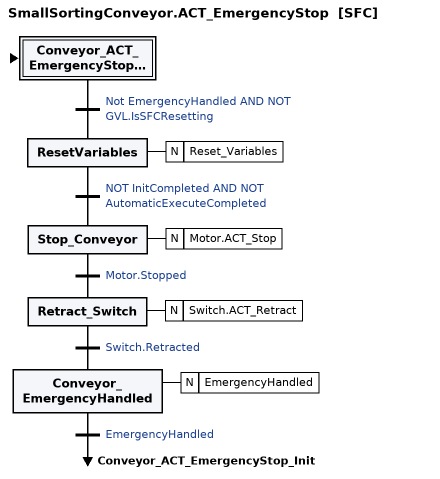
INITIAL_STEP Conveyor_ACT_EmergencyStop_Init:
END_STEP
TRANSITION FROM Conveyor_ACT_EmergencyStop_Init TO ResetVariables
  := Not EmergencyHandled AND NOT GVL.IsSFCResetting;
END_TRANSITION
STEP ResetVariables:
  Reset_Variables(N);
END_STEP
TRANSITION FROM ResetVariables TO Stop_Conveyor
  := NOT InitCompleted AND NOT AutomaticExecuteCompleted;
END_TRANSITION
STEP Stop_Conveyor:
  Motor.ACT_Stop(N);
END_STEP
TRANSITION FROM Stop_Conveyor TO Retract_Switch
  := Motor.Stopped;
END_TRANSITION
STEP Retract_Switch:
  Switch.ACT_Retract(N);
END_STEP
TRANSITION FROM Retract_Switch TO Conveyor_EmergencyHandled
  := Switch.Retracted;
END_TRANSITION
STEP Conveyor_EmergencyHandled:
  EmergencyHandled(N);
END_STEP
TRANSITION FROM Conveyor_EmergencyHandled TO Conveyor_ACT_EmergencyStop_Init
  := EmergencyHandled;
END_TRANSITION
END_ACTION

ACTION ACT_Init:
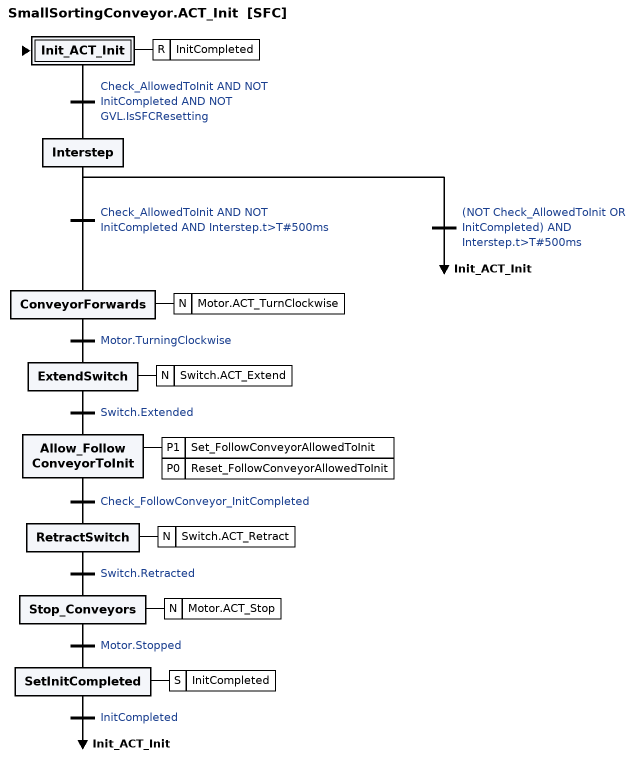
INITIAL_STEP Init_ACT_Init:
  InitCompleted(R);
END_STEP
TRANSITION FROM Init_ACT_Init TO Interstep
  := Check_AllowedToInit AND NOT InitCompleted AND NOT GVL.IsSFCResetting;
END_TRANSITION
STEP Interstep:
END_STEP
TRANSITION FROM Interstep TO ConveyorForwards
  := Check_AllowedToInit AND NOT InitCompleted AND Interstep.t>T#500ms;
END_TRANSITION
TRANSITION FROM Interstep TO Init_ACT_Init
  := (NOT Check_AllowedToInit OR InitCompleted) AND Interstep.t>T#500ms;
END_TRANSITION
STEP ConveyorForwards:
  Motor.ACT_TurnClockwise(N);
END_STEP
TRANSITION FROM ConveyorForwards TO ExtendSwitch
  := Motor.TurningClockwise;
END_TRANSITION
STEP ExtendSwitch:
  Switch.ACT_Extend(N);
END_STEP
TRANSITION FROM ExtendSwitch TO Allow_FollowConveyorToInit
  := Switch.Extended;
END_TRANSITION
STEP Allow_FollowConveyorToInit:
  Set_FollowConveyorAllowedToInit(P1);
  Reset_FollowConveyorAllowedToInit(P0);
END_STEP
TRANSITION FROM Allow_FollowConveyorToInit TO RetractSwitch
  := Check_FollowConveyor_InitCompleted;
END_TRANSITION
STEP RetractSwitch:
  Switch.ACT_Retract(N);
END_STEP
TRANSITION FROM RetractSwitch TO Stop_Conveyors
  := Switch.Retracted;
END_TRANSITION
STEP Stop_Conveyors:
  Motor.ACT_Stop(N);
END_STEP
TRANSITION FROM Stop_Conveyors TO SetInitCompleted
  := Motor.Stopped;
END_TRANSITION
STEP SetInitCompleted:
  InitCompleted(S);
END_STEP
TRANSITION FROM SetInitCompleted TO Init_ACT_Init
  := InitCompleted;
END_TRANSITION
END_ACTION
END_FUNCTION_BLOCK

FUNCTION_BLOCK Stack
VAR_INPUT	
	//Hardware
	Seperator : MonostableCylinder;
	Panel : OperationPanel;	
	WPAvailable : MicroSwitch;
	InductiveSensor : InductiveSensor;
	OpticalSensor : OpticalSensor;
	WeightModule : WeightModule;
	
	//Software
	Check_WPPickedUp : BOOL;
	SFCReset : BOOL;	//Only for SFC implementation
END_VAR
VAR_OUTPUT	
	//Software
	StartButton : BOOL;
	ManuelMode : BOOL;
	AutomaticMode : BOOL;
	InitCompleted : BOOL;
	AutomaticExecuteCompleted : BOOL;
	EmergencyStop : BOOL;
	EmergencyHandled : BOOL;	
	
END_VAR
VAR	
	//Software
	WPProvided : BOOL;	
	WPType_White : BOOL;
	WPType_Black : BOOL;
	WPType_Metallic : BOOL;	
	WPWeight_Light : BOOL;
	WPWeight_Medium : BOOL;
	WPWeight_Heavy : BOOL;	
	Timer : TON;	
END_VAR

                  Panel();
StartButton := Panel.StartButton;
ManuelMode := Panel.ManuelMode; 
AutomaticMode := Panel.AutomaticMode;
EmergencyStop := Panel.EmergencyStop;
Check_WPPickedUp := Main.Check_Stack_WPPickedUp;
                

ACTION Reset_Timer:
                      Timer(IN:=FALSE);
                    
END_ACTION

ACTION Reset_Variables:
                      InitCompleted := FALSE;
AutomaticExecuteCompleted := FALSE;

WPType_White:=FALSE;
WPType_Black:=FALSE;
WPType_Metallic:=FALSE;
WPWeight_Light:=FALSE;
WPWeight_Medium:=FALSE;
WPWeight_Heavy:=FALSE;
                    
END_ACTION

ACTION Set_Timer250ms:
                      Timer(IN:=TRUE, PT:=T#250MS);
                    
END_ACTION

ACTION Set_WPParameters_AND_WPProvided:
                      //WPType
IF(NOT InductiveSensor.DI_WPMetallic AND NOT OpticalSensor.DI_WPLight)THEN
	WPType_Black:=TRUE;
	WPType_White:=FALSE;
	WPType_Metallic:=FALSE;
ELSIF(NOT InductiveSensor.DI_WPMetallic AND OpticalSensor.DI_WPLight)THEN
	WPType_Black:=FALSE;
	WPType_White:=TRUE;
	WPType_Metallic:=FALSE;
ELSIF(InductiveSensor.DI_WPMetallic)THEN
	WPType_Black:=FALSE;
	WPType_White:=FALSE;
	WPType_Metallic:=TRUE;
END_IF
//WPWeight
IF(WeightModule.AI_WPWeight<12000)THEN
	WPWeight_Light:=TRUE;
	WPWeight_Medium:=FALSE;
	WPWeight_Heavy:=FALSE;
ELSIF(12000<=WeightModule.AI_WPWeight AND WeightModule.AI_WPWeight<24000)THEN
	WPWeight_Light:=FALSE;
	WPWeight_Medium:=TRUE;
	WPWeight_Heavy:=FALSE;
ELSIF(2400<=WeightModule.AI_WPWeight)THEN
	WPWeight_Light:=FALSE;
	WPWeight_Medium:=FALSE;
	WPWeight_Heavy:=TRUE;	
END_IF

WPProvided:=TRUE;
                    
END_ACTION

ACTION ACT_ProvideWP:
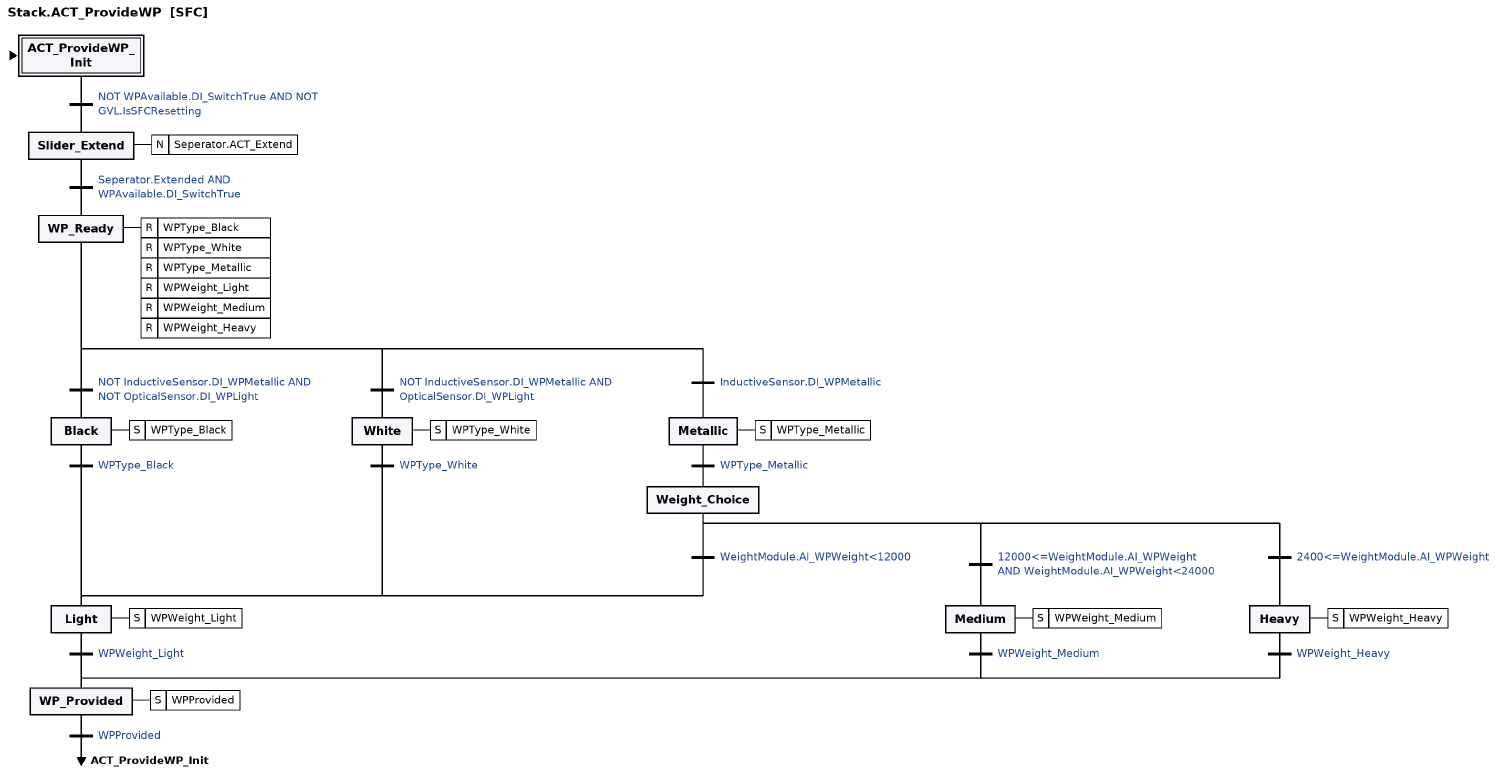
INITIAL_STEP ACT_ProvideWP_Init:
END_STEP
TRANSITION FROM ACT_ProvideWP_Init TO Slider_Extend
  := NOT WPAvailable.DI_SwitchTrue AND NOT GVL.IsSFCResetting;
END_TRANSITION
STEP Slider_Extend:
  Seperator.ACT_Extend(N);
END_STEP
TRANSITION FROM Slider_Extend TO WP_Ready
  := Seperator.Extended AND WPAvailable.DI_SwitchTrue;
END_TRANSITION
STEP WP_Ready:
  WPType_Black(R);
  WPType_White(R);
  WPType_Metallic(R);
  WPWeight_Light(R);
  WPWeight_Medium(R);
  WPWeight_Heavy(R);
END_STEP
TRANSITION FROM WP_Ready TO Black
  := NOT InductiveSensor.DI_WPMetallic AND NOT OpticalSensor.DI_WPLight;
END_TRANSITION
TRANSITION FROM WP_Ready TO White
  := NOT InductiveSensor.DI_WPMetallic AND OpticalSensor.DI_WPLight;
END_TRANSITION
TRANSITION FROM WP_Ready TO Metallic
  := InductiveSensor.DI_WPMetallic;
END_TRANSITION
STEP Black:
  WPType_Black(S);
END_STEP
TRANSITION FROM Black TO Light
  := WPType_Black;
END_TRANSITION
STEP Light:
  WPWeight_Light(S);
END_STEP
TRANSITION FROM Light TO WP_Provided
  := WPWeight_Light;
END_TRANSITION
STEP White:
  WPType_White(S);
END_STEP
TRANSITION FROM White TO Light
  := WPType_White;
END_TRANSITION
STEP Metallic:
  WPType_Metallic(S);
END_STEP
TRANSITION FROM Metallic TO Weight_Choice
  := WPType_Metallic;
END_TRANSITION
STEP Weight_Choice:
END_STEP
TRANSITION FROM Weight_Choice TO Light
  := WeightModule.AI_WPWeight<12000;
END_TRANSITION
TRANSITION FROM Weight_Choice TO Medium
  := 12000<=WeightModule.AI_WPWeight AND WeightModule.AI_WPWeight<24000;
END_TRANSITION
TRANSITION FROM Weight_Choice TO Heavy
  := 2400<=WeightModule.AI_WPWeight;
END_TRANSITION
STEP Medium:
  WPWeight_Medium(S);
END_STEP
TRANSITION FROM Medium TO WP_Provided
  := WPWeight_Medium;
END_TRANSITION
STEP Heavy:
  WPWeight_Heavy(S);
END_STEP
TRANSITION FROM Heavy TO WP_Provided
  := WPWeight_Heavy;
END_TRANSITION
STEP WP_Provided:
  WPProvided(S);
END_STEP
TRANSITION FROM WP_Provided TO ACT_ProvideWP_Init
  := WPProvided;
END_TRANSITION
END_ACTION

ACTION ACT_AutomaticExecute:
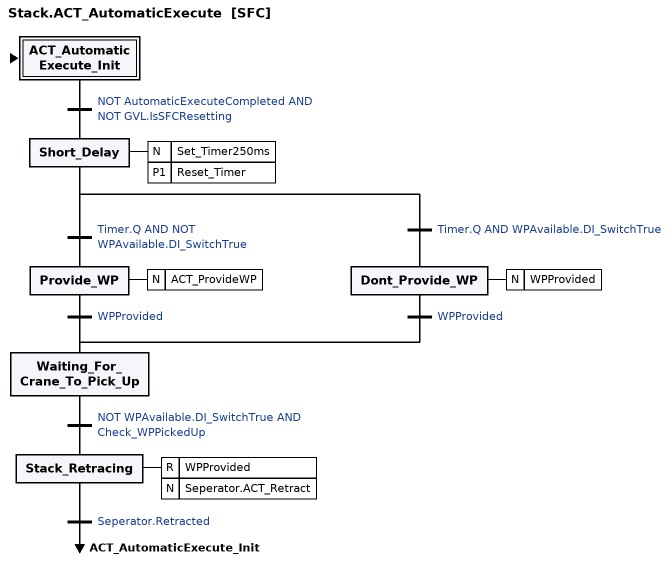
INITIAL_STEP ACT_AutomaticExecute_Init:
END_STEP
TRANSITION FROM ACT_AutomaticExecute_Init TO Short_Delay
  := NOT AutomaticExecuteCompleted AND NOT GVL.IsSFCResetting;
END_TRANSITION
STEP Short_Delay:
  Set_Timer250ms(N);
  Reset_Timer(P1);
END_STEP
TRANSITION FROM Short_Delay TO Provide_WP
  := Timer.Q AND NOT WPAvailable.DI_SwitchTrue;
END_TRANSITION
TRANSITION FROM Short_Delay TO Dont_Provide_WP
  := Timer.Q AND WPAvailable.DI_SwitchTrue;
END_TRANSITION
STEP Provide_WP:
  ACT_ProvideWP(N);
END_STEP
TRANSITION FROM Provide_WP TO Waiting_For_Crane_To_Pick_Up
  := WPProvided;
END_TRANSITION
STEP Dont_Provide_WP:
  WPProvided(N);
END_STEP
TRANSITION FROM Dont_Provide_WP TO Waiting_For_Crane_To_Pick_Up
  := WPProvided;
END_TRANSITION
STEP Waiting_For_Crane_To_Pick_Up:
END_STEP
TRANSITION FROM Waiting_For_Crane_To_Pick_Up TO Stack_Retracing
  := NOT WPAvailable.DI_SwitchTrue AND Check_WPPickedUp;
END_TRANSITION
STEP Stack_Retracing:
  WPProvided(R);
  Seperator.ACT_Retract(N);
END_STEP
TRANSITION FROM Stack_Retracing TO ACT_AutomaticExecute_Init
  := Seperator.Retracted;
END_TRANSITION
END_ACTION

ACTION ACT_EmergencyStop:
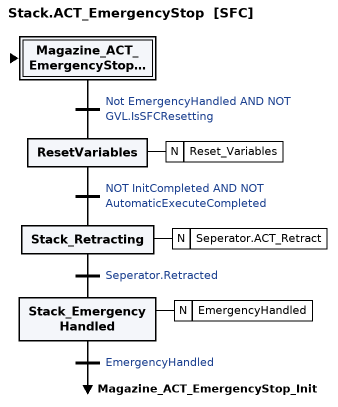
INITIAL_STEP Magazine_ACT_EmergencyStop_Init:
END_STEP
TRANSITION FROM Magazine_ACT_EmergencyStop_Init TO ResetVariables
  := Not EmergencyHandled AND NOT GVL.IsSFCResetting;
END_TRANSITION
STEP ResetVariables:
  Reset_Variables(N);
END_STEP
TRANSITION FROM ResetVariables TO Stack_Retracting
  := NOT InitCompleted AND NOT AutomaticExecuteCompleted;
END_TRANSITION
STEP Stack_Retracting:
  Seperator.ACT_Retract(N);
END_STEP
TRANSITION FROM Stack_Retracting TO Stack_EmergencyHandled
  := Seperator.Retracted;
END_TRANSITION
STEP Stack_EmergencyHandled:
  EmergencyHandled(N);
END_STEP
TRANSITION FROM Stack_EmergencyHandled TO Magazine_ACT_EmergencyStop_Init
  := EmergencyHandled;
END_TRANSITION
END_ACTION

ACTION ACT_Init:
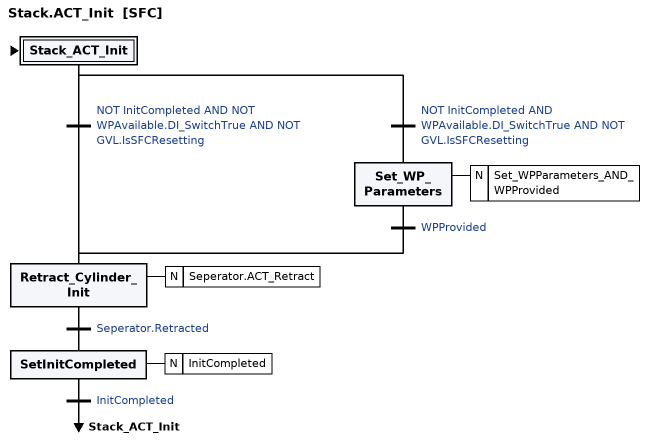
INITIAL_STEP Stack_ACT_Init:
END_STEP
TRANSITION FROM Stack_ACT_Init TO Retract_Cylinder_Init
  := NOT InitCompleted AND NOT WPAvailable.DI_SwitchTrue AND NOT GVL.IsSFCResetting;
END_TRANSITION
TRANSITION FROM Stack_ACT_Init TO Set_WP_Parameters
  := NOT InitCompleted AND WPAvailable.DI_SwitchTrue AND NOT GVL.IsSFCResetting;
END_TRANSITION
STEP Set_WP_Parameters:
  Set_WPParameters_AND_WPProvided(N);
END_STEP
TRANSITION FROM Set_WP_Parameters TO Retract_Cylinder_Init
  := WPProvided;
END_TRANSITION
STEP Retract_Cylinder_Init:
  Seperator.ACT_Retract(N);
END_STEP
TRANSITION FROM Retract_Cylinder_Init TO SetInitCompleted
  := Seperator.Retracted;
END_TRANSITION
STEP SetInitCompleted:
  InitCompleted(N);
END_STEP
TRANSITION FROM SetInitCompleted TO Stack_ACT_Init
  := InitCompleted;
END_TRANSITION
END_ACTION
END_FUNCTION_BLOCK

FUNCTION_BLOCK Stamp
VAR_INPUT
	//Hardware
	Panel : OperationPanel;
	PressureSensor : PressureSensor;
	PropValve : ProportionalValve;
	WPAvailable : MicroSwitch;
	StampingCylinder : MonostableCylinder;
	SlidingCylinder : BistableCylinder;			
	
	//Software	
	SoftwareEmergency : BOOL;
	Check_Allowed_To_Operate : BOOL;
	Check_WPWeight_Light : BOOL;
	Check_WPWeight_Medium : BOOL;
    Check_WPWeight_Heavy : BOOL;
	SFCReset : BOOL;	//Only for SFC implementation
END_VAR
VAR_OUTPUT
	//Software
	StartButton : BOOL;	
	ManuelMode : BOOL;
	AutomaticMode : BOOL;
	InitCompleted : BOOL;
	AutomaticExecuteCompleted : BOOL;
	EmergencyStop : BOOL;		
	EmergencyHandled : BOOL;
	IsStamping : BOOL;
	
END_VAR
VAR
	//Software
	WPStamped : BOOL;
	WPType_White : BOOL;
	WPType_Black : BOOL;
	WPType_Metallic : BOOL;
	WPWeight_Light : BOOL;
	WPWeight_Medium : BOOL;
	WPWeight_Heavy : BOOL;
	Timer : TON;	
END_VAR

                  Panel();
StartButton := Panel.StartButton;
ManuelMode := Panel.ManuelMode; 
AutomaticMode := Panel.AutomaticMode;
EmergencyStop := Panel.EmergencyStop;
Check_Allowed_To_Operate := Main.Check_Stamp_AllowedToOperate;
Check_WPWeight_Light:=Main.Crane_WPWeight_Light;
Check_WPWeight_Medium:=Main.Crane_WPWeight_Medium;
Check_WPWeight_Heavy:=Main.Crane_WPWeight_Heavy;
                

ACTION ExtendStampingCylinder_AND_Timer1500ms:
                      StampingCylinder.ACT_Extend();
Timer(IN:=TRUE, PT:=T#1500MS);
                    
END_ACTION

ACTION Reset_Pressure:
                      PropValve.AO_SetPressure:=0;
                    
END_ACTION

ACTION Reset_Timer:
                      Timer(IN:=FALSE);
                    
END_ACTION

ACTION Reset_Variables:
                      InitCompleted := FALSE;
AutomaticExecuteCompleted := FALSE;

propValve.AO_SetPressure:=0;
IsStamping:=FALSE;
WPStamped:=FALSE;
WPType_Black := FALSE;
WPType_White := FALSE;
WPType_Metallic := FALSE;
WPWeight_Light := FALSE;
WPWeight_Medium := FALSE;
WPWeight_Heavy := FALSE;
                    
END_ACTION

ACTION Set_HeavyPressure:
                      PropValve.AO_SetPressure:=7000;
                    
END_ACTION

ACTION Set_LightPressure:
                      PropValve.AO_SetPressure:=4000;
                    
END_ACTION

ACTION Set_MediumPressure:
                      PropValve.AO_SetPressure:=5500;
                    
END_ACTION

ACTION Set_Timer1000ms:
                      Timer(IN:=TRUE, PT:=T#1000MS);
                    
END_ACTION

ACTION Set_Timer500ms:
                      Timer(IN:=TRUE, PT:=T#500ms);
                    
END_ACTION

ACTION Set_WPWeight:
                      WPWeight_Light := Check_WPWeight_Light;
WPWeight_Medium := Check_WPWeight_Medium;
WPWeight_Heavy := Check_WPWeight_Heavy;
                    
END_ACTION

ACTION ACT_Stamp:
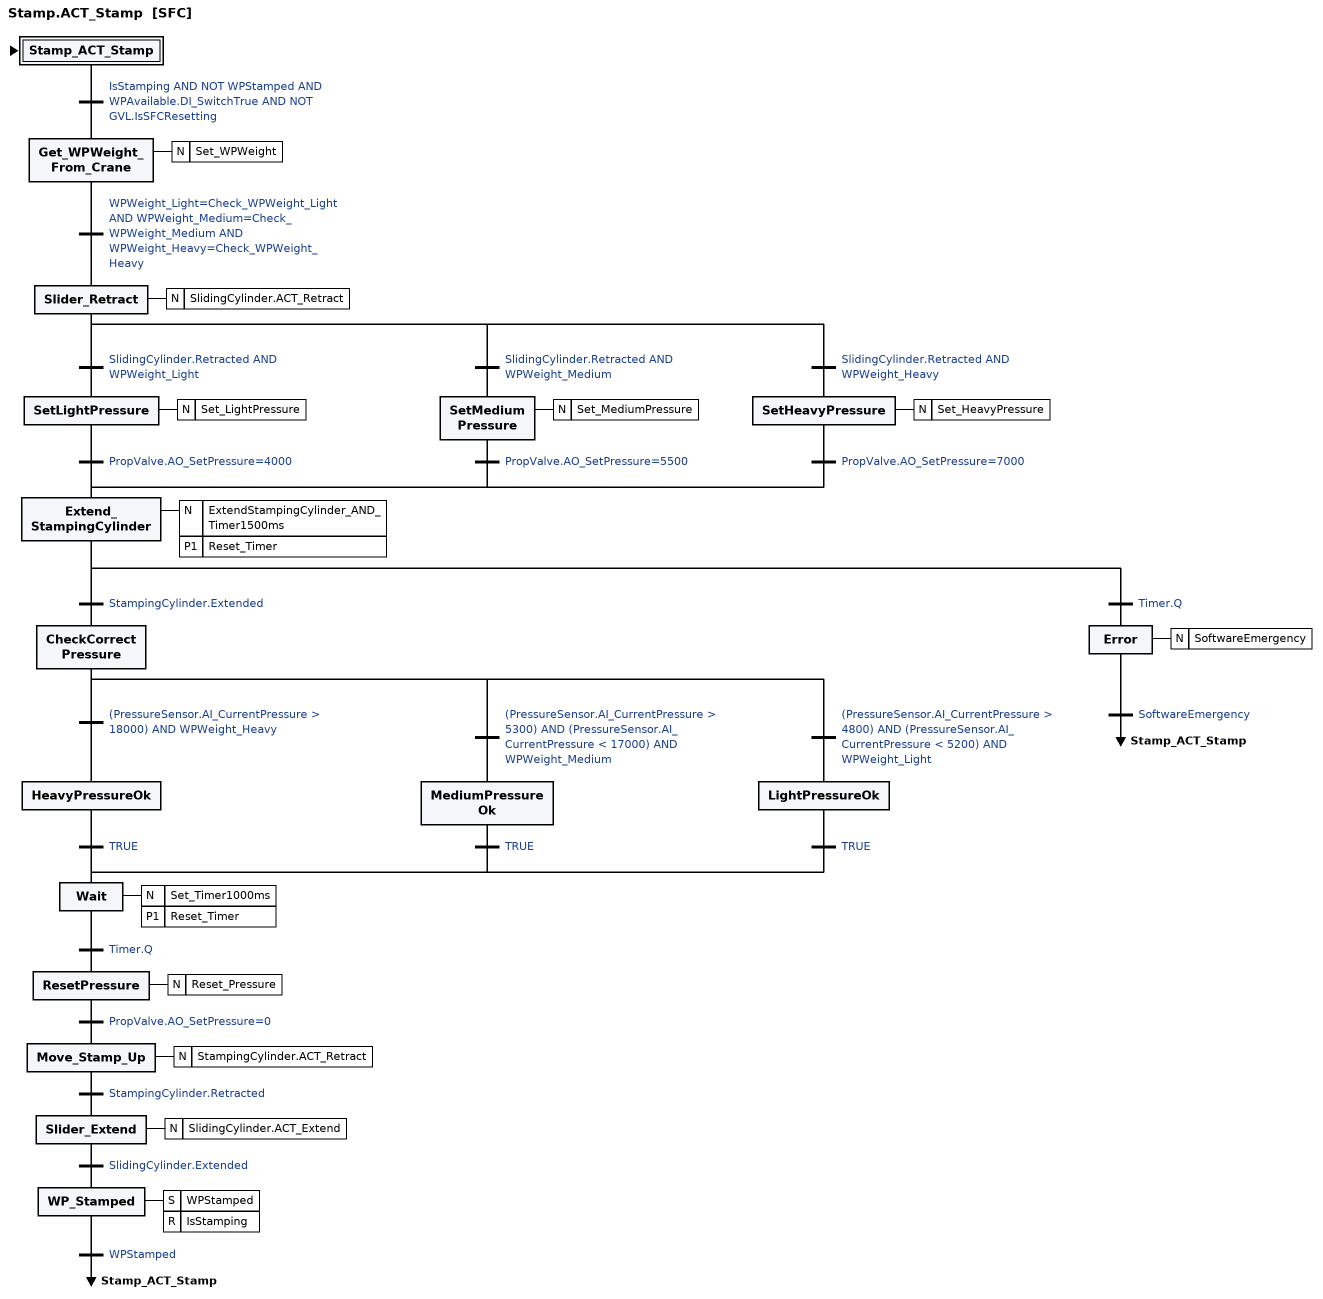
INITIAL_STEP Stamp_ACT_Stamp:
END_STEP
TRANSITION FROM Stamp_ACT_Stamp TO Get_WPWeight_From_Crane
  := IsStamping AND NOT WPStamped AND WPAvailable.DI_SwitchTrue AND NOT GVL.IsSFCResetting;
END_TRANSITION
STEP Get_WPWeight_From_Crane:
  Set_WPWeight(N);
END_STEP
TRANSITION FROM Get_WPWeight_From_Crane TO Slider_Retract
  := WPWeight_Light=Check_WPWeight_Light AND WPWeight_Medium=Check_WPWeight_Medium AND WPWeight_Heavy=Check_WPWeight_Heavy;
END_TRANSITION
STEP Slider_Retract:
  SlidingCylinder.ACT_Retract(N);
END_STEP
TRANSITION FROM Slider_Retract TO SetLightPressure
  := SlidingCylinder.Retracted AND WPWeight_Light;
END_TRANSITION
TRANSITION FROM Slider_Retract TO SetMediumPressure
  := SlidingCylinder.Retracted AND WPWeight_Medium;
END_TRANSITION
TRANSITION FROM Slider_Retract TO SetHeavyPressure
  := SlidingCylinder.Retracted AND WPWeight_Heavy;
END_TRANSITION
STEP SetLightPressure:
  Set_LightPressure(N);
END_STEP
TRANSITION FROM SetLightPressure TO Extend_StampingCylinder
  := PropValve.AO_SetPressure=4000;
END_TRANSITION
STEP SetMediumPressure:
  Set_MediumPressure(N);
END_STEP
TRANSITION FROM SetMediumPressure TO Extend_StampingCylinder
  := PropValve.AO_SetPressure=5500;
END_TRANSITION
STEP SetHeavyPressure:
  Set_HeavyPressure(N);
END_STEP
TRANSITION FROM SetHeavyPressure TO Extend_StampingCylinder
  := PropValve.AO_SetPressure=7000;
END_TRANSITION
STEP Extend_StampingCylinder:
  ExtendStampingCylinder_AND_Timer1500ms(N);
  Reset_Timer(P1);
END_STEP
TRANSITION FROM Extend_StampingCylinder TO CheckCorrectPressure
  := StampingCylinder.Extended;
END_TRANSITION
TRANSITION FROM Extend_StampingCylinder TO Error
  := Timer.Q;
END_TRANSITION
STEP CheckCorrectPressure:
END_STEP
TRANSITION FROM CheckCorrectPressure TO HeavyPressureOk
  := (PressureSensor.AI_CurrentPressure > 18000) AND WPWeight_Heavy;
END_TRANSITION
TRANSITION FROM CheckCorrectPressure TO MediumPressureOk
  := (PressureSensor.AI_CurrentPressure > 5300) AND (PressureSensor.AI_CurrentPressure < 17000) AND WPWeight_Medium;
END_TRANSITION
TRANSITION FROM CheckCorrectPressure TO LightPressureOk
  := (PressureSensor.AI_CurrentPressure > 4800) AND (PressureSensor.AI_CurrentPressure < 5200) AND WPWeight_Light;
END_TRANSITION
STEP HeavyPressureOk:
END_STEP
TRANSITION FROM HeavyPressureOk TO Wait
  := TRUE;
END_TRANSITION
STEP MediumPressureOk:
END_STEP
TRANSITION FROM MediumPressureOk TO Wait
  := TRUE;
END_TRANSITION
STEP LightPressureOk:
END_STEP
TRANSITION FROM LightPressureOk TO Wait
  := TRUE;
END_TRANSITION
STEP Error:
  SoftwareEmergency(N);
END_STEP
TRANSITION FROM Error TO Stamp_ACT_Stamp
  := SoftwareEmergency;
END_TRANSITION
STEP Wait:
  Set_Timer1000ms(N);
  Reset_Timer(P1);
END_STEP
TRANSITION FROM Wait TO ResetPressure
  := Timer.Q;
END_TRANSITION
STEP ResetPressure:
  Reset_Pressure(N);
END_STEP
TRANSITION FROM ResetPressure TO Move_Stamp_Up
  := PropValve.AO_SetPressure=0;
END_TRANSITION
STEP Move_Stamp_Up:
  StampingCylinder.ACT_Retract(N);
END_STEP
TRANSITION FROM Move_Stamp_Up TO Slider_Extend
  := StampingCylinder.Retracted;
END_TRANSITION
STEP Slider_Extend:
  SlidingCylinder.ACT_Extend(N);
END_STEP
TRANSITION FROM Slider_Extend TO WP_Stamped
  := SlidingCylinder.Extended;
END_TRANSITION
STEP WP_Stamped:
  WPStamped(S);
  IsStamping(R);
END_STEP
TRANSITION FROM WP_Stamped TO Stamp_ACT_Stamp
  := WPStamped;
END_TRANSITION
END_ACTION

ACTION ACT_AutomaticExecute:
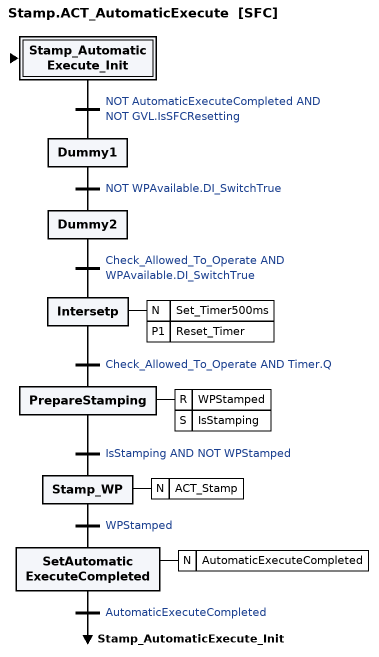
INITIAL_STEP Stamp_AutomaticExecute_Init:
END_STEP
TRANSITION FROM Stamp_AutomaticExecute_Init TO Dummy1
  := NOT AutomaticExecuteCompleted AND NOT GVL.IsSFCResetting;
END_TRANSITION
STEP Dummy1:
END_STEP
TRANSITION FROM Dummy1 TO Dummy2
  := NOT WPAvailable.DI_SwitchTrue;
END_TRANSITION
STEP Dummy2:
END_STEP
TRANSITION FROM Dummy2 TO Intersetp
  := Check_Allowed_To_Operate AND WPAvailable.DI_SwitchTrue;
END_TRANSITION
STEP Intersetp:
  Set_Timer500ms(N);
  Reset_Timer(P1);
END_STEP
TRANSITION FROM Intersetp TO PrepareStamping
  := Check_Allowed_To_Operate AND Timer.Q;
END_TRANSITION
STEP PrepareStamping:
  WPStamped(R);
  IsStamping(S);
END_STEP
TRANSITION FROM PrepareStamping TO Stamp_WP
  := IsStamping AND NOT WPStamped;
END_TRANSITION
STEP Stamp_WP:
  ACT_Stamp(N);
END_STEP
TRANSITION FROM Stamp_WP TO SetAutomaticExecuteCompleted
  := WPStamped;
END_TRANSITION
STEP SetAutomaticExecuteCompleted:
  AutomaticExecuteCompleted(N);
END_STEP
TRANSITION FROM SetAutomaticExecuteCompleted TO Stamp_AutomaticExecute_Init
  := AutomaticExecuteCompleted;
END_TRANSITION
END_ACTION

ACTION ACT_EmergencyStop:
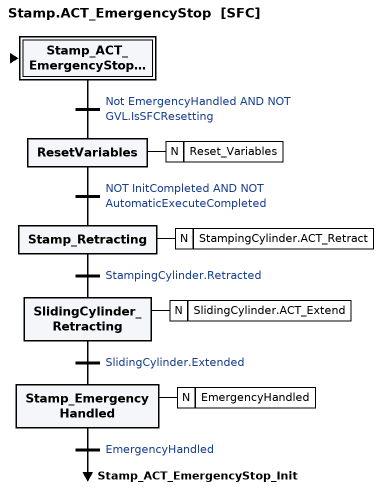
INITIAL_STEP Stamp_ACT_EmergencyStop_Init:
END_STEP
TRANSITION FROM Stamp_ACT_EmergencyStop_Init TO ResetVariables
  := Not EmergencyHandled AND NOT GVL.IsSFCResetting;
END_TRANSITION
STEP ResetVariables:
  Reset_Variables(N);
END_STEP
TRANSITION FROM ResetVariables TO Stamp_Retracting
  := NOT InitCompleted AND NOT AutomaticExecuteCompleted;
END_TRANSITION
STEP Stamp_Retracting:
  StampingCylinder.ACT_Retract(N);
END_STEP
TRANSITION FROM Stamp_Retracting TO SlidingCylinder_Retracting
  := StampingCylinder.Retracted;
END_TRANSITION
STEP SlidingCylinder_Retracting:
  SlidingCylinder.ACT_Extend(N);
END_STEP
TRANSITION FROM SlidingCylinder_Retracting TO Stamp_EmergencyHandled
  := SlidingCylinder.Extended;
END_TRANSITION
STEP Stamp_EmergencyHandled:
  EmergencyHandled(N);
END_STEP
TRANSITION FROM Stamp_EmergencyHandled TO Stamp_ACT_EmergencyStop_Init
  := EmergencyHandled;
END_TRANSITION
END_ACTION

ACTION ACT_Init:
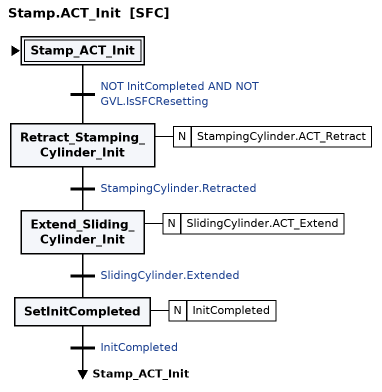
INITIAL_STEP Stamp_ACT_Init:
END_STEP
TRANSITION FROM Stamp_ACT_Init TO Retract_Stamping_Cylinder_Init
  := NOT InitCompleted AND NOT GVL.IsSFCResetting;
END_TRANSITION
STEP Retract_Stamping_Cylinder_Init:
  StampingCylinder.ACT_Retract(N);
END_STEP
TRANSITION FROM Retract_Stamping_Cylinder_Init TO Extend_Sliding_Cylinder_Init
  := StampingCylinder.Retracted;
END_TRANSITION
STEP Extend_Sliding_Cylinder_Init:
  SlidingCylinder.ACT_Extend(N);
END_STEP
TRANSITION FROM Extend_Sliding_Cylinder_Init TO SetInitCompleted
  := SlidingCylinder.Extended;
END_TRANSITION
STEP SetInitCompleted:
  InitCompleted(N);
END_STEP
TRANSITION FROM SetInitCompleted TO Stamp_ACT_Init
  := InitCompleted;
END_TRANSITION
END_ACTION
END_FUNCTION_BLOCK

FUNCTION_BLOCK PPU
VAR_INPUT	
	//Hardware
	Stack : Stack;		
	Crane : Crane;	
	LargeSortingConveyor : LargeSortingConveyor;	
	Stamp : Stamp;	
	PicAlphaConveyor : PicAlphaConveyor;
	SmallSortingConveyor : SmallSortingConveyor;
	RefillConveyor : RefillConveyor;
	PicAlpha : PicAlpha;
	SafetyDoor : SafetyDoor; 
	LightGrid : LightGrid;
	
	//Software
	SFCReset : BOOL; //Only for SFC implementation
END_VAR
VAR_OUTPUT
	//Software	
	StartButton : BOOL;
	ManuelMode : BOOL;
	AutomaticMode : BOOL;
	InitCompleted : BOOL;	
	AutomaticExecuteCompleted : BOOL;
	EmergencyStop : BOOL;
	EmergencyHandled : BOOL;
	SFCResetResetCompleted : BOOL;	//Only for SFC implementation
	SFCResetCompleted : BOOL; //Only for SFC implementation
END_VAR
VAR	
	Timer : TON;
	t : time := T#1500ms;
END_VAR

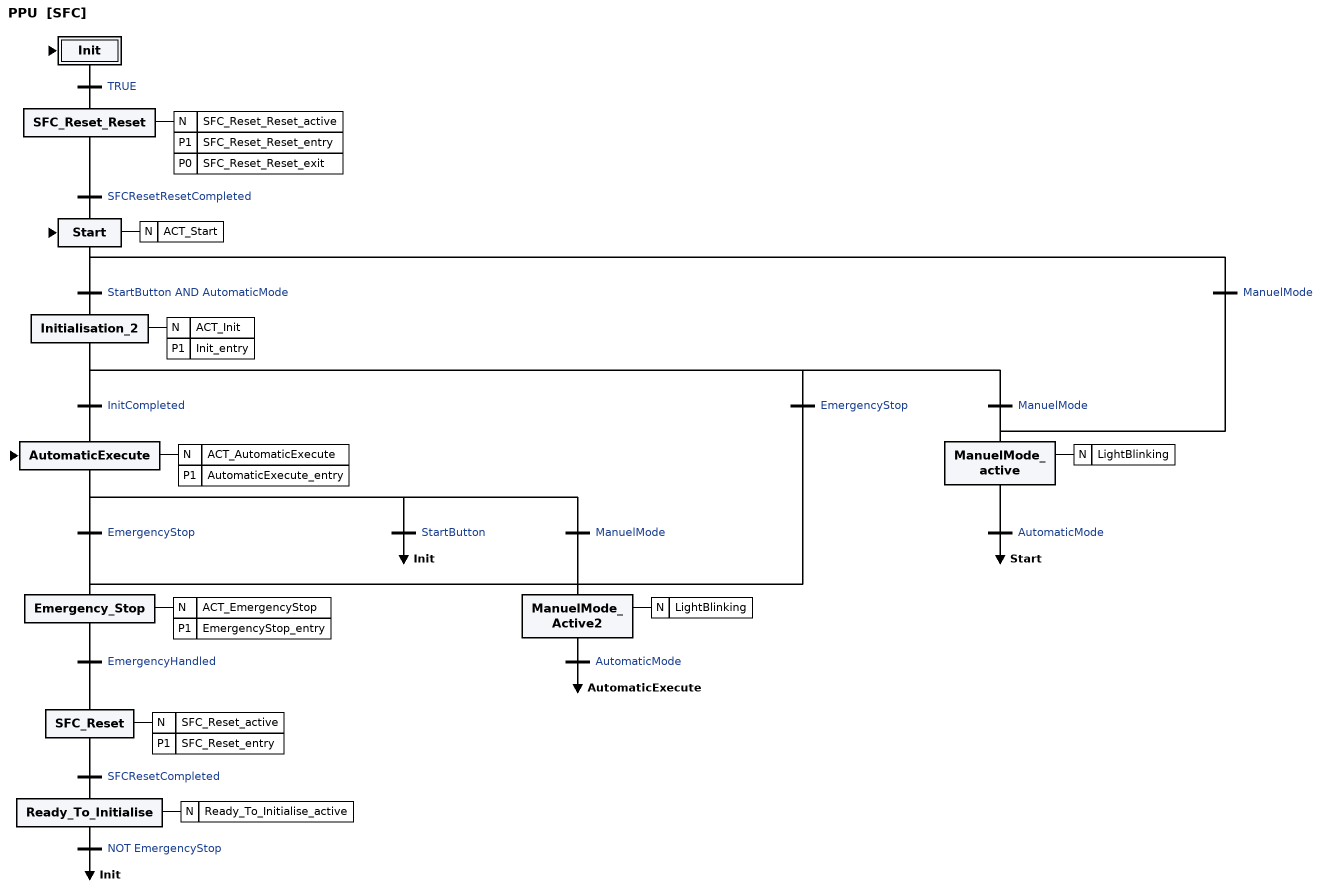
INITIAL_STEP Init:
END_STEP
TRANSITION FROM Init TO SFC_Reset_Reset
  := TRUE;
END_TRANSITION
STEP SFC_Reset_Reset:
  SFC_Reset_Reset_active(N);
  SFC_Reset_Reset_entry(P1);
  SFC_Reset_Reset_exit(P0);
END_STEP
TRANSITION FROM SFC_Reset_Reset TO Start
  := SFCResetResetCompleted;
END_TRANSITION
STEP Start:
  ACT_Start(N);
END_STEP
TRANSITION FROM Start TO Initialisation_2
  := StartButton AND AutomaticMode;
END_TRANSITION
TRANSITION FROM Start TO ManuelMode_active
  := ManuelMode;
END_TRANSITION
STEP ManuelMode_active:
  LightBlinking(N);
END_STEP
TRANSITION FROM ManuelMode_active TO Start
  := AutomaticMode;
END_TRANSITION
STEP Initialisation_2:
  ACT_Init(N);
  Init_entry(P1);
END_STEP
TRANSITION FROM Initialisation_2 TO AutomaticExecute
  := InitCompleted;
END_TRANSITION
TRANSITION FROM Initialisation_2 TO Emergency_Stop
  := EmergencyStop;
END_TRANSITION
TRANSITION FROM Initialisation_2 TO ManuelMode_active
  := ManuelMode;
END_TRANSITION
STEP AutomaticExecute:
  ACT_AutomaticExecute(N);
  AutomaticExecute_entry(P1);
END_STEP
TRANSITION FROM AutomaticExecute TO Emergency_Stop
  := EmergencyStop;
END_TRANSITION
TRANSITION FROM AutomaticExecute TO Init
  := StartButton;
END_TRANSITION
TRANSITION FROM AutomaticExecute TO ManuelMode_Active2
  := ManuelMode;
END_TRANSITION
STEP ManuelMode_Active2:
  LightBlinking(N);
END_STEP
TRANSITION FROM ManuelMode_Active2 TO AutomaticExecute
  := AutomaticMode;
END_TRANSITION
STEP Emergency_Stop:
  ACT_EmergencyStop(N);
  EmergencyStop_entry(P1);
END_STEP
TRANSITION FROM Emergency_Stop TO SFC_Reset
  := EmergencyHandled;
END_TRANSITION
STEP SFC_Reset:
  SFC_Reset_active(N);
  SFC_Reset_entry(P1);
END_STEP
TRANSITION FROM SFC_Reset TO Ready_To_Initialise
  := SFCResetCompleted;
END_TRANSITION
STEP Ready_To_Initialise:
  Ready_To_Initialise_active(N);
END_STEP
TRANSITION FROM Ready_To_Initialise TO Init
  := NOT EmergencyStop;
END_TRANSITION

ACTION ACT_CheckEmergency:
                      EmergencyStop := Stack.EmergencyStop OR LargeSortingConveyor.EmergencyStop OR Stamp.EmergencyStop OR SafetyDoor.EmergencyStop OR LightGrid.EmergencyStop OR Crane.SoftwareEmergency OR Stamp.SoftwareEmergency OR PicAlpha.SoftwareEmergency;
                    
END_ACTION

ACTION ACT_CheckManuelMode:
                      ManuelMode := Stack.ManuelMode OR LargeSortingConveyor.ManuelMode OR Stamp.ManuelMode OR SafetyDoor.ManuelMode OR LightGrid.ManuelMode;
AutomaticMode := Stack.AutomaticMode AND LargeSortingConveyor.AutomaticMode AND Stamp.AutomaticMode AND SafetyDoor.AutomaticMode AND LightGrid.AutomaticMode;
                    
END_ACTION

ACTION ACT_Start:
                      StartButton := Stack.StartButton OR LargeSortingConveyor.StartButton OR Stamp.StartButton OR SafetyDoor.StartButton OR LightGrid.StartButton;
ManuelMode := Stack.ManuelMode OR LargeSortingConveyor.ManuelMode OR Stamp.ManuelMode OR SafetyDoor.ManuelMode OR LightGrid.ManuelMode;
AutomaticMode := Stack.AutomaticMode AND LargeSortingConveyor.AutomaticMode AND Stamp.AutomaticMode AND SafetyDoor.AutomaticMode AND LightGrid.AutomaticMode;
                    
END_ACTION

ACTION AutomaticExecute_entry:
                      AutomaticExecuteCompleted:=FALSE;

LargeSortingConveyor.Panel.ACT_TurnLampWhite_Off();
Stack.Panel.ACT_TurnLampWhite_Off();	
Stamp.Panel.ACT_TurnLampWhite_Off();
LargeSortingConveyor.Panel.ACT_TurnLampGreen_On();
Stack.Panel.ACT_TurnLampGreen_On();	
Stamp.Panel.ACT_TurnLampGreen_On();
                    
END_ACTION

ACTION CallAll_AutomationExecutes:
                      EmergencyStop := Stack.EmergencyStop OR LargeSortingConveyor.EmergencyStop OR Stamp.EmergencyStop OR SafetyDoor.EmergencyStop OR LightGrid.EmergencyStop OR Crane.SoftwareEmergency OR Stamp.SoftwareEmergency OR PicAlpha.SoftwareEmergency;
StartButton := Stack.StartButton OR LargeSortingConveyor.StartButton OR Stamp.StartButton OR SafetyDoor.StartButton OR LightGrid.StartButton;
ManuelMode := Stack.ManuelMode OR LargeSortingConveyor.ManuelMode OR Stamp.ManuelMode OR SafetyDoor.ManuelMode OR LightGrid.ManuelMode;
AutomaticMode := Stack.AutomaticMode AND LargeSortingConveyor.AutomaticMode AND Stamp.AutomaticMode AND SafetyDoor.AutomaticMode AND LightGrid.AutomaticMode;
Crane.ACT_AutomaticExecute();
Stack.ACT_AutomaticExecute();
Stamp.ACT_AutomaticExecute();
LargeSortingConveyor.ACT_AutomaticExecute();
PicAlphaConveyor.ACT_AutomaticExecute();
SmallSortingConveyor.ACT_AutomaticExecute();
RefillConveyor.ACT_AutomaticExecute();
PicAlpha.ACT_AutomaticExecute();
                    
END_ACTION

ACTION EmergencyStop_entry:
                      EmergencyHandled:=FALSE;

LargeSortingConveyor.Panel.ACT_TurnLampWhite_Off();
Stack.Panel.ACT_TurnLampWhite_Off();	
Stamp.Panel.ACT_TurnLampWhite_Off();
LargeSortingConveyor.Panel.ACT_TurnLampGreen_Off();
Stack.Panel.ACT_TurnLampGreen_Off();	
Stamp.Panel.ACT_TurnLampGreen_Off();
                    
END_ACTION

ACTION Init_entry:
                      InitCompleted:=FALSE;

LargeSortingConveyor.Panel.ACT_TurnLampWhite_On();
Stack.Panel.ACT_TurnLampWhite_On();	
Stamp.Panel.ACT_TurnLampWhite_On();
LargeSortingConveyor.Panel.ACT_TurnLampGreen_Off();
Stack.Panel.ACT_TurnLampGreen_Off();	
Stamp.Panel.ACT_TurnLampGreen_Off();
                    
END_ACTION

ACTION LightBlinking:
                      Timer(IN := NOT Timer.Q, PT:=t);

IF (Timer.ET < Timer.PT/2) THEN
	//GREEN
	Stack.Panel.ACT_TurnLampGreen_On();
	LargeSortingConveyor.Panel.ACT_TurnLampGreen_On();
	Stamp.Panel.ACT_TurnLampGreen_On();
	SafetyDoor.Panel.ACT_TurnLampGreen_On();
	LightGrid.Panel.ACT_TurnLampGreen_On();
	Stack.Panel.ACT_TurnLampWhite_Off();
	LargeSortingConveyor.Panel.ACT_TurnLampWhite_Off();	
	Stamp.Panel.ACT_TurnLampWhite_Off();
	SafetyDoor.Panel.ACT_TurnLampReset_Off();
	LightGrid.Panel.ACT_TurnLampReset_Off();
ELSE
	//WHITE
	Stack.Panel.ACT_TurnLampGreen_Off();
	LargeSortingConveyor.Panel.ACT_TurnLampGreen_Off();
	Stamp.Panel.ACT_TurnLampGreen_Off();
	SafetyDoor.Panel.ACT_TurnLampGreen_Off();
	LightGrid.Panel.ACT_TurnLampGreen_Off();
	Stack.Panel.ACT_TurnLampWhite_On();
	LargeSortingConveyor.Panel.ACT_TurnLampWhite_On();	
	Stamp.Panel.ACT_TurnLampWhite_On();
	SafetyDoor.Panel.ACT_TurnLampReset_On();
	LightGrid.Panel.ACT_TurnLampReset_On();
END_IF

AutomaticMode := Stack.AutomaticMode AND LargeSortingConveyor.AutomaticMode AND Stamp.AutomaticMode AND SafetyDoor.AutomaticMode AND LightGrid.AutomaticMode;
                    
END_ACTION

ACTION Ready_To_Initialise_active:
                      EmergencyStop := Stack.EmergencyStop OR LargeSortingConveyor.EmergencyStop OR Stamp.EmergencyStop OR SafetyDoor.EmergencyStop OR LightGrid.EmergencyStop OR Crane.SoftwareEmergency OR Stamp.SoftwareEmergency OR PicAlpha.SoftwareEmergency;
StartButton := Stack.StartButton OR LargeSortingConveyor.StartButton OR Stamp.StartButton OR SafetyDoor.StartButton OR LightGrid.StartButton;
IF(StartButton)THEN
	Stamp.SoftwareEmergency:=FALSE;
	Crane.SoftwareEmergency:=FALSE;
	PicAlpha.SoftwareEmergency:=FALSE;
END_IF	
                    
END_ACTION

ACTION SFC_Reset_active:
                      (*PPU*)
	//Variables
	InitCompleted:=FALSE;
	AutomaticExecuteCompleted:=FALSE;

(*Crane Reset*)
	Crane(SFCReset:=TRUE);
	Crane.ACT_Init(SFCReset:=TRUE);
	Crane.ACT_AutomaticExecute(SFCReset:=TRUE);
	Crane.ACT_EmergencyStop(SFCReset:=TRUE);
	Crane.ACT_MoveToConveyor(SFCReset:=TRUE);
	Crane.ACT_MoveToStack(SFCReset:=TRUE);
	Crane.ACT_MoveToStamp(SFCReset:=TRUE);
	Crane.ACT_PickUpWP(SFCReset:=TRUE);
	Crane.ACT_PutDownWP(SFCReset:=TRUE);

(*LargeSortingConveyor Reset*)
	LargeSortingConveyor(SFCReset:=TRUE);
	LargeSortingConveyor.ACT_Init(SFCReset:=TRUE);
	LargeSortingConveyor.ACT_AutomaticExecute(SFCReset:=TRUE);
	LargeSortingConveyor.ACT_ChangeTarget(SFCReset:=TRUE);
	LargeSortingConveyor.ACT_CheckWPType(SFCReset:=TRUE);	
	LargeSortingConveyor.ACT_SortWP(SFCReset:=TRUE);
	
(*Stack Reset*)
	Stack(SFCReset:=TRUE);
	Stack.ACT_Init(SFCReset:=TRUE);
	Stack.ACT_AutomaticExecute(SFCReset:=TRUE);
	Stack.ACT_ProvideWP(SFCReset:=TRUE);

(*Stamp Reset*)
	Stamp(SFCReset:=TRUE);
	Stamp.ACT_Init(SFCReset:=TRUE);
	Stamp.ACT_AutomaticExecute(SFCReset:=TRUE);
	Stamp.ACT_Stamp(SFCReset:=TRUE);
	
(*PicAlphaConveyor Reset*)
	PicAlphaConveyor(SFCReset:=TRUE);
	PicAlphaConveyor.ACT_Init(SFCReset:=TRUE);
	PicAlphaConveyor.ACT_AutomaticExecute(SFCReset:=TRUE);
	PicAlphaConveyor.ACT_SeperateWP(SFCReset:=TRUE);
	
(*SmallSortingConveyor Reset*)
	SmallSortingConveyor(SFCReset:=TRUE); 
	SmallSortingConveyor.ACT_Init(SFCReset:=TRUE);
	SmallSortingConveyor.ACT_AutomaticExecute(SFCReset:=TRUE);
	SmallSortingConveyor.ACT_SortWP(SFCReset:=TRUE);
	SmallSortingConveyor.ACT_ChangeTarget(SFCReset:=TRUE);
	SmallSortingConveyor.ACT_CheckWPType(SFCReset:=TRUE);
	
(*RefillConveyor Reset*)
	RefillConveyor(SFCReset:=TRUE);
	RefillConveyor.ACT_Init(SFCReset:=TRUE);
	RefillConveyor.ACT_AutomaticExecute(SFCReset:=TRUE);
	RefillConveyor.ACT_SeperateWP(SFCReset:=TRUE);
	
(*PicAlpha Reset*)
	PicAlpha(SFCReset:=TRUE);
	PicAlpha.ACT_Init(SFCReset:=TRUE);
	PicAlpha.ACT_AutomaticExecute(SFCReset:=TRUE);
	PicAlpha.ACT_MoveToPos1(SFCReset:=TRUE);
	PicAlpha.ACT_MoveToPos2(SFCReset:=TRUE);
	PicAlpha.ACT_MoveToPos3(SFCReset:=TRUE);
	PicAlpha.ACT_MoveToPos4(SFCReset:=TRUE);
	PicAlpha.ACT_PickUpWP(SFCReset:=TRUE);
	PicAlpha.ACT_PutDownWP(SFCReset:=TRUE);
	
SFCResetCompleted:=TRUE;	
                    
END_ACTION

ACTION SFC_Reset_entry:
                      SFCResetCompleted:=FALSE;
GVL.IsSFCResetting:=TRUE;
                    
END_ACTION

ACTION SFC_Reset_Reset_active:
                      (*Crane Reset*)	
	Crane(SFCReset:=FALSE);
	Crane.ACT_Init(SFCReset:=FALSE);							
	Crane.ACT_AutomaticExecute(SFCReset:=FALSE);				
	Crane.ACT_EmergencyStop(SFCReset:=FALSE);					
	Crane.ACT_MoveToConveyor(SFCReset:=FALSE);					
	Crane.ACT_MoveToStack(SFCReset:=FALSE);						
	Crane.ACT_MoveToStamp(SFCReset:=FALSE);						
	Crane.ACT_PickUpWP(SFCReset:=FALSE);						
	Crane.ACT_PutDownWP(SFCReset:=FALSE);
	Crane.LiftingCylinder.ACT_Retract();
	Crane.Gripper.ACT_Release();
	Crane.Table.Motor.ACT_Stop();	
	//Variables
	Crane.SFCReset:=FALSE;
	
                                                               
(*LargeSortingConveyor Reset*)  
	LargeSortingConveyor(SFCReset:=FALSE);                                
	LargeSortingConveyor.ACT_Init(SFCReset:=FALSE);				
	LargeSortingConveyor.ACT_AutomaticExecute(SFCReset:=FALSE);	
	LargeSortingConveyor.ACT_ChangeTarget(SFCReset:=FALSE);		
	LargeSortingConveyor.ACT_CheckWPType(SFCReset:=FALSE);		
	LargeSortingConveyor.ACT_SortWP(SFCReset:=FALSE);	
	LargeSortingConveyor.Motor.ACT_Stop();
	LargeSortingConveyor.Seperator1.ACT_Retract();
	LargeSortingConveyor.Seperator2.ACT_Retract();
	//Variables
	LargeSortingConveyor.SFCReset:=FALSE;
	                                                            
(*Stack Reset*)   
	Stack(SFCReset:=FALSE);                                              
	Stack.ACT_Init(SFCReset:=FALSE);							
	Stack.ACT_AutomaticExecute(SFCReset:=FALSE);				
	Stack.ACT_ProvideWP(SFCReset:=FALSE);	
	Stack.Seperator.ACT_Retract();
	//Variables	
	Stack.SFCReset:=FALSE;
                                                        
(*Stamp Reset*)  
	Stamp(SFCReset:=FALSE);                                               
	Stamp.ACT_Init(SFCReset:=FALSE);							
	Stamp.ACT_AutomaticExecute(SFCReset:=FALSE);				
	Stamp.ACT_Stamp(SFCReset:=FALSE);
	Stamp.StampingCylinder.ACT_Retract();
	Stamp.SlidingCylinder.ACT_Extend();
	//Variables	
	Stamp.SFCReset:=FALSE;

(*PicAlphaConveyor Reset*)
	PicAlphaConveyor(SFCReset:=FALSE); 
	PicAlphaConveyor.ACT_Init(SFCReset:=FALSE);
	PicAlphaConveyor.ACT_AutomaticExecute(SFCReset:=FALSE);
	PicAlphaConveyor.ACT_SeperateWP(SFCReset:=FALSE);
	//Variables
	PicAlphaConveyor.SFCReset:=FALSE;
	
(*SmallSortingConveyor Reset*)
	SmallSortingConveyor(SFCReset:=FALSE); 
	SmallSortingConveyor.ACT_Init(SFCReset:=FALSE);
	SmallSortingConveyor.ACT_AutomaticExecute(SFCReset:=FALSE);
	SmallSortingConveyor.ACT_SortWP(SFCReset:=FALSE);
	SmallSortingConveyor.ACT_ChangeTarget(SFCReset:=FALSE);
	SmallSortingConveyor.ACT_CheckWPType(SFCReset:=FALSE);
	//Variables
	SmallSortingConveyor.SFCReset:=FALSE;
	
(*RefillConveyor Reset*)
	RefillConveyor(SFCReset:=FALSE); 
	RefillConveyor.ACT_Init(SFCReset:=FALSE);
	RefillConveyor.ACT_AutomaticExecute(SFCReset:=FALSE);
	RefillConveyor.ACT_SeperateWP(SFCReset:=FALSE);
	//Variables
	RefillConveyor.SFCReset:=FALSE;	
	
(*PicAlpha Reset*)
	PicAlpha(SFCReset:=FALSE);
	PicAlpha.ACT_Init(SFCReset:=FALSE);
	PicAlpha.ACT_AutomaticExecute(SFCReset:=FALSE);
	PicAlpha.ACT_MoveToPos1(SFCReset:=FALSE);
	PicAlpha.ACT_MoveToPos2(SFCReset:=FALSE);
	PicAlpha.ACT_MoveToPos3(SFCReset:=FALSE);
	PicAlpha.ACT_MoveToPos4(SFCReset:=FALSE);
	PicAlpha.ACT_PickUpWP(SFCReset:=FALSE);
	PicAlpha.ACT_PutDownWP(SFCReset:=FALSE);
	//Variables
	PicAlpha.SFCReset:=FALSE;	
	                                                            
SFCResetResetCompleted:=TRUE;
SFCResetCompleted:=TRUE;
                    
END_ACTION

ACTION SFC_Reset_Reset_entry:
                      SFCResetResetCompleted:=FALSE;
GVL.IsSFCResetting:=TRUE;
                    
END_ACTION

ACTION SFC_Reset_Reset_exit:
                      GVL.IsSFCResetting:=FALSE;
                    
END_ACTION

ACTION ACT_AutomaticExecute:
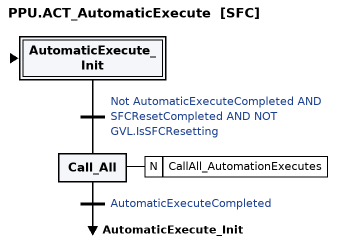
INITIAL_STEP AutomaticExecute_Init:
END_STEP
TRANSITION FROM AutomaticExecute_Init TO Call_All
  := Not AutomaticExecuteCompleted AND SFCResetCompleted AND NOT GVL.IsSFCResetting;
END_TRANSITION
STEP Call_All:
  CallAll_AutomationExecutes(N);
END_STEP
TRANSITION FROM Call_All TO AutomaticExecute_Init
  := AutomaticExecuteCompleted;
END_TRANSITION
END_ACTION

ACTION ACT_EmergencyStop:
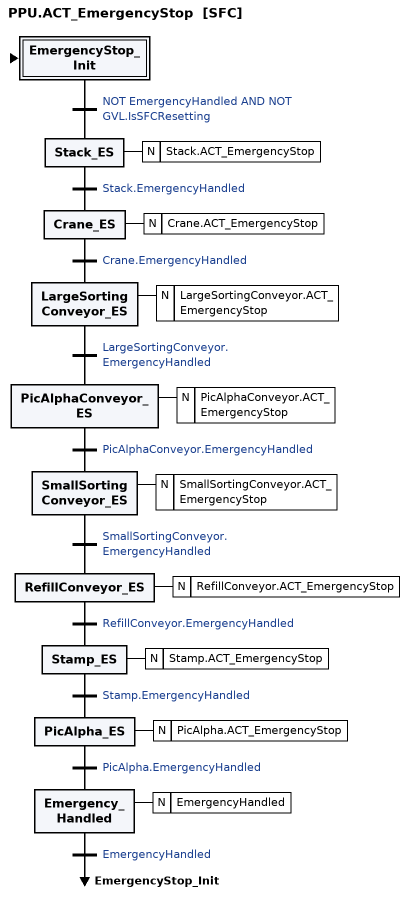
INITIAL_STEP EmergencyStop_Init:
END_STEP
TRANSITION FROM EmergencyStop_Init TO Stack_ES
  := NOT EmergencyHandled AND NOT GVL.IsSFCResetting;
END_TRANSITION
STEP Stack_ES:
  Stack.ACT_EmergencyStop(N);
END_STEP
TRANSITION FROM Stack_ES TO Crane_ES
  := Stack.EmergencyHandled;
END_TRANSITION
STEP Crane_ES:
  Crane.ACT_EmergencyStop(N);
END_STEP
TRANSITION FROM Crane_ES TO LargeSortingConveyor_ES
  := Crane.EmergencyHandled;
END_TRANSITION
STEP LargeSortingConveyor_ES:
  LargeSortingConveyor.ACT_EmergencyStop(N);
END_STEP
TRANSITION FROM LargeSortingConveyor_ES TO PicAlphaConveyor_ES
  := LargeSortingConveyor.EmergencyHandled;
END_TRANSITION
STEP PicAlphaConveyor_ES:
  PicAlphaConveyor.ACT_EmergencyStop(N);
END_STEP
TRANSITION FROM PicAlphaConveyor_ES TO SmallSortingConveyor_ES
  := PicAlphaConveyor.EmergencyHandled;
END_TRANSITION
STEP SmallSortingConveyor_ES:
  SmallSortingConveyor.ACT_EmergencyStop(N);
END_STEP
TRANSITION FROM SmallSortingConveyor_ES TO RefillConveyor_ES
  := SmallSortingConveyor.EmergencyHandled;
END_TRANSITION
STEP RefillConveyor_ES:
  RefillConveyor.ACT_EmergencyStop(N);
END_STEP
TRANSITION FROM RefillConveyor_ES TO Stamp_ES
  := RefillConveyor.EmergencyHandled;
END_TRANSITION
STEP Stamp_ES:
  Stamp.ACT_EmergencyStop(N);
END_STEP
TRANSITION FROM Stamp_ES TO PicAlpha_ES
  := Stamp.EmergencyHandled;
END_TRANSITION
STEP PicAlpha_ES:
  PicAlpha.ACT_EmergencyStop(N);
END_STEP
TRANSITION FROM PicAlpha_ES TO Emergency_Handled
  := PicAlpha.EmergencyHandled;
END_TRANSITION
STEP Emergency_Handled:
  EmergencyHandled(N);
END_STEP
TRANSITION FROM Emergency_Handled TO EmergencyStop_Init
  := EmergencyHandled;
END_TRANSITION
END_ACTION

ACTION ACT_Init:
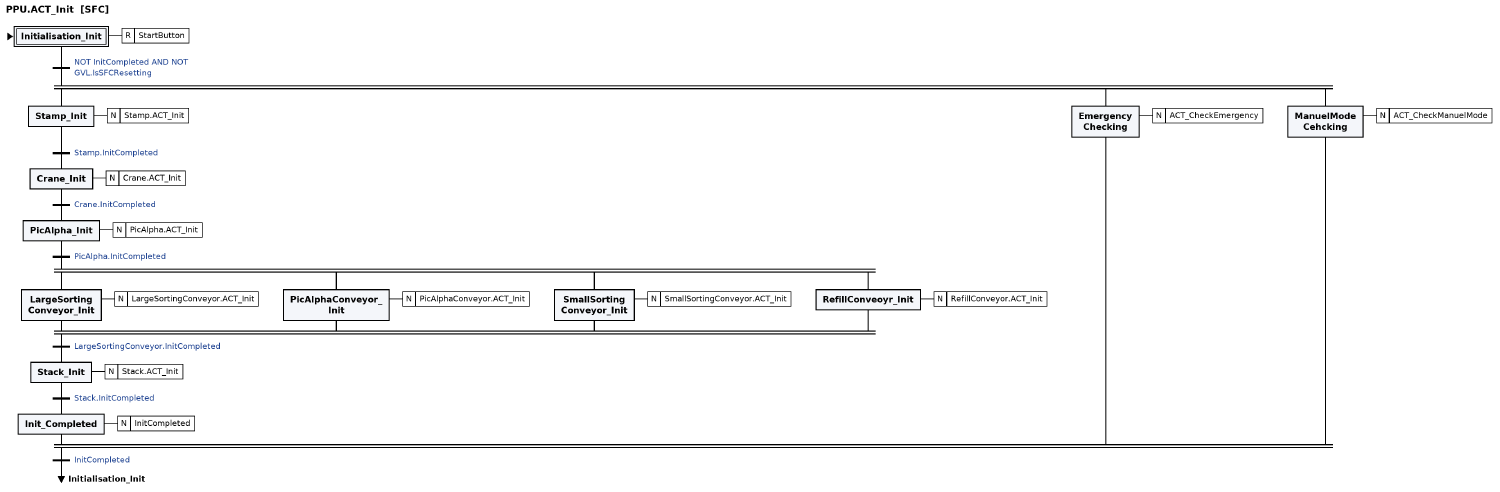
INITIAL_STEP Initialisation_Init:
  StartButton(R);
END_STEP
TRANSITION FROM Initialisation_Init TO (Stamp_Init, EmergencyChecking, ManuelModeCehcking)
  := NOT InitCompleted AND NOT GVL.IsSFCResetting;
END_TRANSITION
STEP Stamp_Init:
  Stamp.ACT_Init(N);
END_STEP
TRANSITION FROM Stamp_Init TO Crane_Init
  := Stamp.InitCompleted;
END_TRANSITION
STEP Crane_Init:
  Crane.ACT_Init(N);
END_STEP
TRANSITION FROM Crane_Init TO PicAlpha_Init
  := Crane.InitCompleted;
END_TRANSITION
STEP PicAlpha_Init:
  PicAlpha.ACT_Init(N);
END_STEP
TRANSITION FROM PicAlpha_Init TO (LargeSortingConveyor_Init, PicAlphaConveyor_Init, SmallSortingConveyor_Init, RefillConveoyr_Init)
  := PicAlpha.InitCompleted;
END_TRANSITION
STEP LargeSortingConveyor_Init:
  LargeSortingConveyor.ACT_Init(N);
END_STEP
TRANSITION FROM (LargeSortingConveyor_Init, PicAlphaConveyor_Init, SmallSortingConveyor_Init, RefillConveoyr_Init) TO Stack_Init
  := LargeSortingConveyor.InitCompleted;
END_TRANSITION
STEP PicAlphaConveyor_Init:
  PicAlphaConveyor.ACT_Init(N);
END_STEP
STEP SmallSortingConveyor_Init:
  SmallSortingConveyor.ACT_Init(N);
END_STEP
STEP RefillConveoyr_Init:
  RefillConveyor.ACT_Init(N);
END_STEP
STEP Stack_Init:
  Stack.ACT_Init(N);
END_STEP
TRANSITION FROM Stack_Init TO Init_Completed
  := Stack.InitCompleted;
END_TRANSITION
STEP Init_Completed:
  InitCompleted(N);
END_STEP
TRANSITION FROM (Init_Completed, EmergencyChecking, ManuelModeCehcking) TO Initialisation_Init
  := InitCompleted;
END_TRANSITION
STEP EmergencyChecking:
  ACT_CheckEmergency(N);
END_STEP
STEP ManuelModeCehcking:
  ACT_CheckManuelMode(N);
END_STEP
END_ACTION
END_FUNCTION_BLOCK

CONFIGURATION Application
  RESOURCE Scenario_19 ON PLC
(* global variable list GVL *)
{attribute 'qualified_only'}
VAR_GLOBAL
	IsSFCResetting : BOOL;
END_VAR
    TASK PlcTask(INTERVAL := T#0ms, PRIORITY := 20);
    PROGRAM MAIN WITH PlcTask : MAIN;
  END_RESOURCE
END_CONFIGURATION
